% RSLogix 500 project minimal_tripper.RSS, saved by version 8.30.00.16 %
PROJECT "UNTITLED"    % processor: Bul.1763 MicroLogix 1100 Series B %

PROGRAM FILES
  LAD 2   5 rungs

DATA FILES
  O0 OUTPUT  4 elements
  I1 INPUT  6 elements
  S2 STATUS  66 elements
  B3 BINARY  1 elements
  T4 TIMER  1 elements
  C5 COUNTER  1 elements
  R6 CONTROL  1 elements
  N7 INTEGER  20 elements
  F8 FLOAT  1 elements

LADDER 2
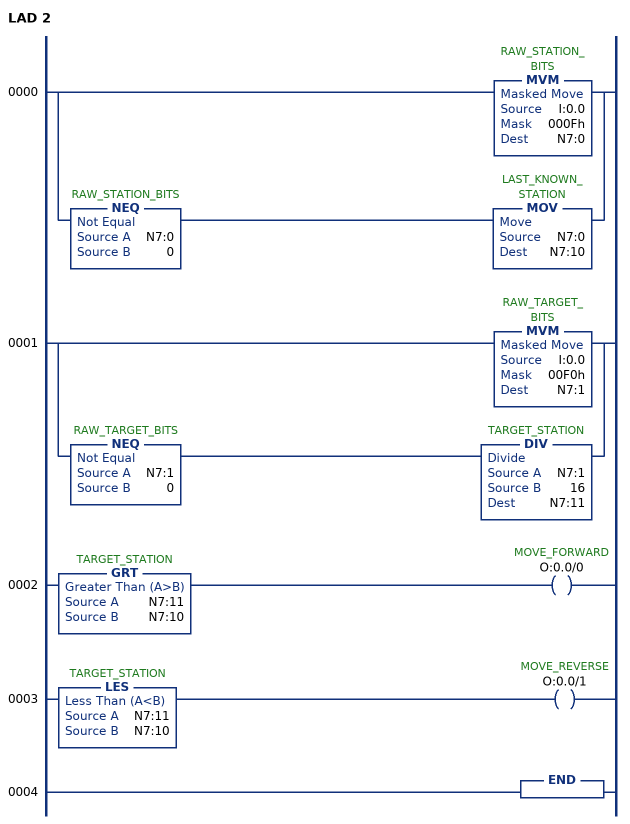
% Rung: 0 %
SOR BST MVM I:0.0 000Fh N7:0 NXB NEQ N7:0 0 MOV N7:0 N7:10 BND EOR
%   N7:0  RAW_STATION_BITS %
%   N7:10  LAST_KNOWN_STATION %
% Rung: 1 %
SOR BST MVM I:0.0 00F0h N7:1 NXB NEQ N7:1 0 DIV N7:1 16 N7:11 BND EOR
%   N7:1  RAW_TARGET_BITS %
%   N7:11  TARGET_STATION %
% Rung: 2 %
SOR GRT N7:11 N7:10 OTE O:0.0/0 EOR
%   N7:11  TARGET_STATION %
%   N7:10  LAST_KNOWN_STATION %
%   O:0.0/0  MOVE_FORWARD %
% Rung: 3 %
SOR LES N7:11 N7:10 OTE O:0.0/1 EOR
%   N7:11  TARGET_STATION %
%   N7:10  LAST_KNOWN_STATION %
%   O:0.0/1  MOVE_REVERSE %
% Rung: 4 %
SOR END EOR

OTHER DOCUMENTED ADDRESSES
  PID  

DATA TABLE (non-zero values as saved)
DATA N7
% N7:10 % 1 1 0 0 0 0 0 0 0 0
